// TIA Portal project "2022.10.15_洗衣机控制系统" (V17)

(* hardware
DEVICE "S7-1200 station_1"  S7-1200 Station
   slot 0: "Rack_0"  S7-1200 Rack  Rack  V1.0
   slot 1: "PLC_1"  CPU 1212C DC/DC/DC  6ES7 212-1AE40-0XB0  V4.5
*)

// ===== PLC "PLC_1"  CPU 1212C DC/DC/DC =====

VAR_GLOBAL   // PLC tag table "默认变量表"
   "System_Byte" AT %MB1 : Byte;
   "FirstScan" AT %M1.0 : Bool;
   "DiagStatusUpdate" AT %M1.1 : Bool;
   "AlwaysTRUE" AT %M1.2 : Bool;
   "AlwaysFALSE" AT %M1.3 : Bool;
END_VAR

VAR_GLOBAL   // PLC tag table "变量表_1"
   "洗衣机启动" AT %I0.0 : Bool;
   "洗衣机停止" AT %I0.1 : Bool;
   "手动排水" AT %I0.2 : Bool;
   "低水位传感器" AT %I0.3 : Bool;
   "高水位传感器" AT %I0.4 : Bool;
   "内部辅助继电器" AT %M0.0 : Bool;
   "进水电磁阀" AT %Q0.0 : Bool;
   "洗机正转" AT %Q0.1 : Bool;
   "洗机反转" AT %Q0.2 : Bool;
   "排水电磁阀" AT %Q0.3 : Bool;
   "脱水电磁离合器" AT %Q0.4 : Bool;
   "完成指示灯" AT %Q0.5 : Bool;
   "定T37" AT %M0.1 : Bool;
   "定T38" AT %M0.2 : Bool;
   "定T39" AT %M0.3 : Bool;
   "定T40" AT %M0.4 : Bool;
   "定T41" AT %M0.5 : Bool;
   "定T42" AT %M0.6 : Bool;
   "计c5" AT %M2.0 : Bool;
   "计c6" AT %M2.1 : Bool;
END_VAR

DATA_BLOCK "定时器"   // DB9
{ S7_Optimized_Access := 'TRUE' }
VERSION : 0.1
   VAR
      T37 : IEC_TIMER;
      T38 : IEC_TIMER;
      T39 : IEC_TIMER;
      T40 : IEC_TIMER;
      T41 : IEC_TIMER;
      T42 : IEC_TIMER;
   END_VAR
BEGIN
END_DATA_BLOCK

// folder: System blocks/Program resources

DATA_BLOCK "T37"   // DB1
{ S7_Optimized_Access := 'TRUE' }
AUTHOR : Simatic
FAMILY : IEC
NAME : IEC_TMR
VERSION : 1.0
// stored: InstanceOfName IEC_TIMER
"IEC_TIMER"
BEGIN
END_DATA_BLOCK

DATA_BLOCK "T38"   // DB2
{ S7_Optimized_Access := 'TRUE' }
AUTHOR : Simatic
FAMILY : IEC
NAME : IEC_TMR
VERSION : 1.0
// stored: InstanceOfName IEC_TIMER
"IEC_TIMER"
BEGIN
END_DATA_BLOCK

DATA_BLOCK "T39"   // DB3
{ S7_Optimized_Access := 'TRUE' }
AUTHOR : Simatic
FAMILY : IEC
NAME : IEC_TMR
VERSION : 1.0
// stored: InstanceOfName IEC_TIMER
"IEC_TIMER"
BEGIN
END_DATA_BLOCK

DATA_BLOCK "T40"   // DB4
{ S7_Optimized_Access := 'TRUE' }
AUTHOR : Simatic
FAMILY : IEC
NAME : IEC_TMR
VERSION : 1.0
// stored: InstanceOfName IEC_TIMER
"IEC_TIMER"
BEGIN
END_DATA_BLOCK

DATA_BLOCK "T41"   // DB5
{ S7_Optimized_Access := 'TRUE' }
AUTHOR : Simatic
FAMILY : IEC
NAME : IEC_TMR
VERSION : 1.0
// stored: InstanceOfName IEC_TIMER
"IEC_TIMER"
BEGIN
END_DATA_BLOCK

DATA_BLOCK "C6"   // DB6
{ S7_Optimized_Access := 'TRUE' }
AUTHOR : Simatic
FAMILY : IEC
NAME : CNTR
VERSION : 1.0
// stored: InstanceOfName IEC_COUNTER
"IEC_COUNTER"
BEGIN
END_DATA_BLOCK

DATA_BLOCK "T42"   // DB7
{ S7_Optimized_Access := 'TRUE' }
AUTHOR : Simatic
FAMILY : IEC
NAME : IEC_TMR
VERSION : 1.0
// stored: InstanceOfName IEC_TIMER
"IEC_TIMER"
BEGIN
END_DATA_BLOCK

DATA_BLOCK "C5"   // DB8
{ S7_Optimized_Access := 'TRUE' }
AUTHOR : Simatic
FAMILY : IEC
NAME : CNTR
VERSION : 1.0
// stored: InstanceOfName IEC_COUNTER
"IEC_COUNTER"
BEGIN
END_DATA_BLOCK

// folder: (top level)

ORGANIZATION_BLOCK "Main"   // OB1, LAD, ProgramCycle
TITLE = "Main Program Sweep (Cycle)"
{ S7_Optimized_Access := 'TRUE' }
VERSION : 0.1
   VAR_INPUT
      Initial_Call : Bool;   // Initial call of this OB
      Remanence : Bool;   // =True, if remanent data are available
   END_VAR
BEGIN

REGION Network 1
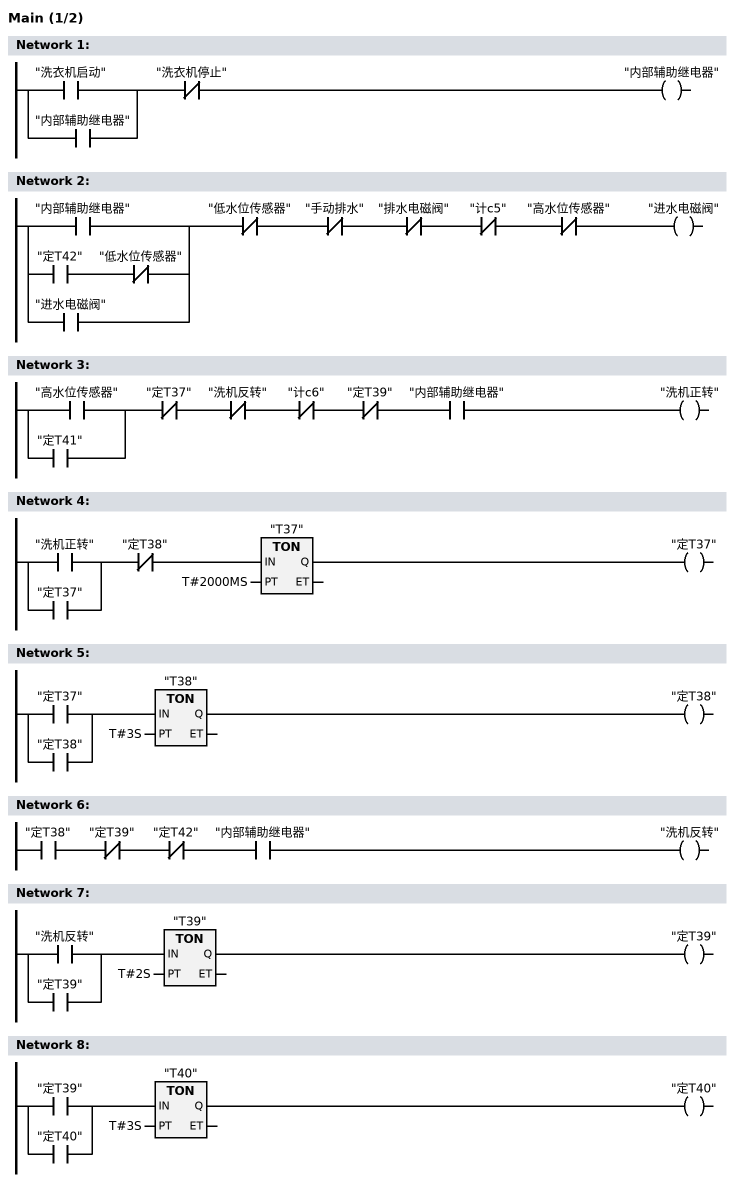
   RUNG wire#powerrail
      Contact( "洗衣机启动" )
      wire#w1
      I_Contact( "洗衣机停止" )
      Coil( "内部辅助继电器" )
   END_RUNG
   RUNG wire#powerrail
      Contact( "内部辅助继电器" )
   END_RUNG wire#w1
   // the same network as SCL:
   "内部辅助继电器" := ("洗衣机启动" OR "内部辅助继电器") AND NOT "洗衣机停止";
END_REGION

REGION Network 2
   RUNG wire#powerrail
      Contact( "内部辅助继电器" )
      wire#w1
      I_Contact( "低水位传感器" )
      I_Contact( "手动排水" )
      I_Contact( "排水电磁阀" )
      I_Contact( "计c5" )
      I_Contact( "高水位传感器" )
      Coil( "进水电磁阀" )
   END_RUNG
   RUNG wire#powerrail
      Contact( "定T42" )
      I_Contact( "低水位传感器" )
   END_RUNG wire#w1
   RUNG wire#powerrail
      Contact( "进水电磁阀" )
   END_RUNG wire#w1
   // the same network as SCL:
   "进水电磁阀" := ("内部辅助继电器" OR ("定T42" AND NOT "低水位传感器") OR "进水电磁阀") AND NOT "低水位传感器" AND NOT "手动排水" AND NOT "排水电磁阀" AND NOT "计c5" AND NOT "高水位传感器";
END_REGION

REGION Network 3
   RUNG wire#powerrail
      Contact( "高水位传感器" )
      wire#w1
      I_Contact( "定T37" )
      I_Contact( "洗机反转" )
      I_Contact( "计c6" )
      I_Contact( "定T39" )
      Contact( "内部辅助继电器" )
      Coil( "洗机正转" )
   END_RUNG
   RUNG wire#powerrail
      Contact( "定T41" )
   END_RUNG wire#w1
   // the same network as SCL:
   "洗机正转" := ("高水位传感器" OR "定T41") AND NOT "定T37" AND NOT "洗机反转" AND NOT "计c6" AND NOT "定T39" AND "内部辅助继电器";
END_REGION

REGION Network 4
   "T37".TON(IN := ("洗机正转" OR "定T37") AND NOT "定T38", PT := T#2000MS);
   "定T37" := "T37".Q;
END_REGION

REGION Network 5
   "T38".TON(IN := "定T37" OR "定T38", PT := T#3S);
   "定T38" := "T38".Q;
END_REGION

REGION Network 6
   RUNG wire#powerrail
      Contact( "定T38" )
      I_Contact( "定T39" )
      I_Contact( "定T42" )
      Contact( "内部辅助继电器" )
      Coil( "洗机反转" )
   END_RUNG
   // the same network as SCL:
   "洗机反转" := "定T38" AND NOT "定T39" AND NOT "定T42" AND "内部辅助继电器";
END_REGION

REGION Network 7
   "T39".TON(IN := "洗机反转" OR "定T39", PT := T#2S);
   "定T39" := "T39".Q;
END_REGION

REGION Network 8
   "T40".TON(IN := "定T39" OR "定T40", PT := T#3S);
   "定T40" := "T40".Q;
END_REGION

REGION Network 9
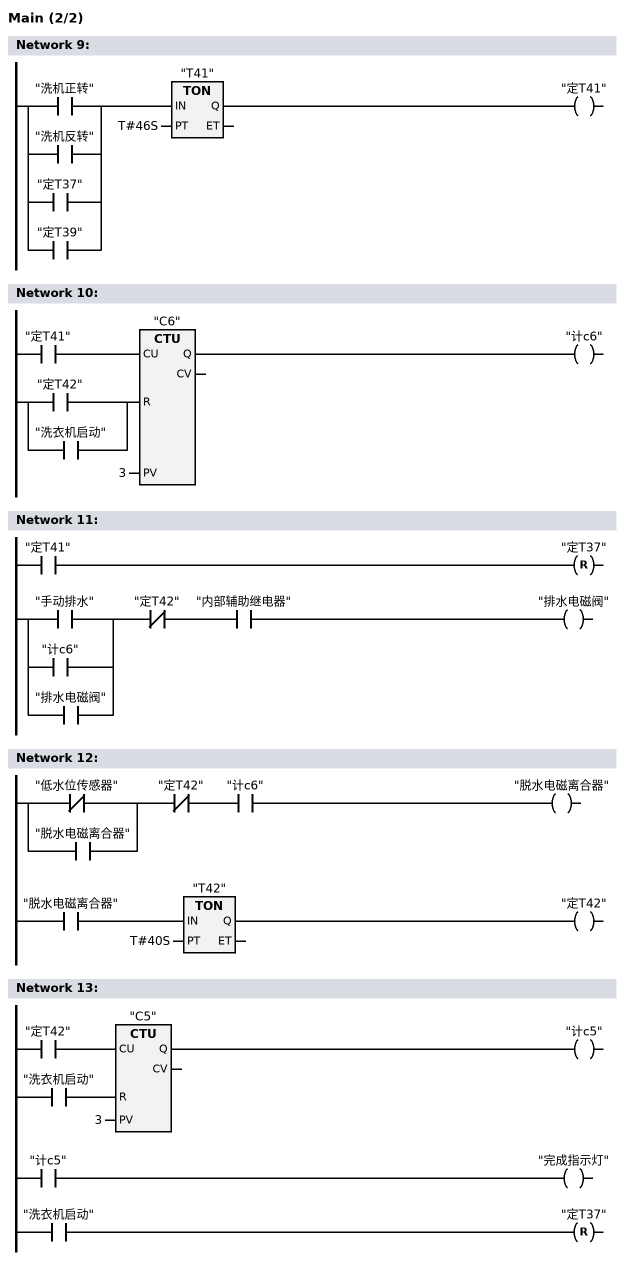
   "T41".TON(IN := "洗机正转" OR "洗机反转" OR "定T37" OR "定T39", PT := T#46S);
   "定T41" := "T41".Q;
END_REGION

REGION Network 10
   "C6".CTU(CU := "定T41", R := "定T42" OR "洗衣机启动", PV := 3);
   "计c6" := "C6".Q;
END_REGION

REGION Network 11
   RUNG wire#powerrail
      Contact( "定T41" )
      R_Coil( "定T37" )
   END_RUNG
   RUNG wire#powerrail
      Contact( "手动排水" )
      wire#w1
      I_Contact( "定T42" )
      Contact( "内部辅助继电器" )
      Coil( "排水电磁阀" )
   END_RUNG
   RUNG wire#powerrail
      Contact( "计c6" )
   END_RUNG wire#w1
   RUNG wire#powerrail
      Contact( "排水电磁阀" )
   END_RUNG wire#w1
   // the same network as SCL:
   IF "定T41" THEN "定T37" := FALSE; END_IF;
   "排水电磁阀" := ("手动排水" OR "计c6" OR "排水电磁阀") AND NOT "定T42" AND "内部辅助继电器";
END_REGION

REGION Network 12
   "脱水电磁离合器" := (NOT "低水位传感器" OR "脱水电磁离合器") AND NOT "定T42" AND "计c6";
   "T42".TON(IN := "脱水电磁离合器", PT := T#40S);
   "定T42" := "T42".Q;
END_REGION

REGION Network 13
   "C5".CTU(CU := "定T42", R := "洗衣机启动", PV := 3);
   "计c5" := "C5".Q;
   "完成指示灯" := "计c5";
   IF "洗衣机启动" THEN "定T37" := FALSE; END_IF;
END_REGION
END_ORGANIZATION_BLOCK